{attribute 'qualified_only'}
{attribute 'strict'}
TYPE E_MMServerStatus :
(
	eMMServerStatus_Default										:= 0,
	eMMServerStatus_Success										:= 1,
	eMMServerStatus_Rejected_UserInputError						:= 2,
	eMMServerStatus_Rejected_NotAllowed							:= 3,
	eMMServerStatus_Rejected_ConfigurationAlreadyDefined		:= 20,
	eMMServerStatus_Rejected_NotDefinedInConfiguration			:= 21,
	eMMServerStatus_Rejected_VehicleRelatedInfoNotFound			:= 40,
	eMMServerStatus_Failed_UnableToRemoveFromConfiguration		:= 100,
	eMMServerStatus_Failed_CouldNotHandleMoveVehicleRequest		:= 120
);
END_TYPE

(* stored: Version 1.1.0.1, ProductVersion 3.1.4024.5
   EnumerationTextList E_MMServerStatus: Id {6fdc5aa4-be99-4219-9f8d-73b6da4b0ad5} *)
